(* IEC 61131-3 sources: ICSQuartz/benchmarks/oscat_basic_upper_case/src, 1 file *)

(* ---- program.st ---- *)
PROGRAM PLC_PRG
VAR_INPUT
    in_STR: STRING;
END_VAR

UPPERCASE(in_STR);

END_PROGRAM
